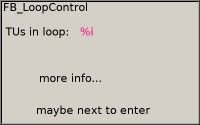
VISUALIZATION V_LoopControl  // 200x125
VAR_IN_OUT
	{attribute 'VAR_IN_OUT_AS_POINTER'}
	fbFunction		: FB_LoopControl;	
END_VAR
    Rectangle (0,0 200x125)
    Label (0,0 200x15), "FB_LoopControl"
    Rectangle (77,22 67x20), "%i", text variable: fbFunction.TuCountInLoop, colour toggle: fbFunction.LoopIsFull
    Label (36,71 92x15), "more info..."
    Label (33,103 123x15), "maybe next to enter"
    Label (4,17 67x30), "TUs in loop:"
END_VISUALIZATION

(* stored: Version 1.1.0.1, ProductVersion 3.1.4024.9
   Visu V_LoopControl: Id {a8edb417-08e2-476b-8ec5-0d7f1f39da80} *)
